// TIA Portal project "四层电梯_V17" (V17)

(* hardware
DEVICE "S7-1200 station_1"  S7-1200 Station
   slot 0: "Rack_0"  S7-1200 Rack  Rack  V1.0
   slot 1: "PLC_1"  CPU 1214C DC/DC/DC  6ES7 214-1AG40-0XB0  V4.2
DEVICE "HMI_1"  KTP700 Basic PN
   slot 0: "HMI_1"  KTP700 Basic PN  6AV2 123-2GB03-0AX0  15.0.0.0
   slot 1: "HMI_RT_1"  KTP700 Basic PN  6AV2 123-2GB03-0AX0  15.0.0.0
   slot 5: "HMI_1.IE_CP_1"  PROFINET Interface  15.0.0.0
      slot 1: "PROFINET Interface_1"  PROFINET Interface
         slot 1: "Port_1"  Port
*)

// ===== PLC "PLC_1"  CPU 1214C DC/DC/DC =====

VAR_GLOBAL   // PLC tag table "默认变量表"
   "System_Byte" AT %MB1 : Byte;
   "FirstScan" AT %M1.0 : Bool;
   "DiagStatusUpdate" AT %M1.1 : Bool;
   "AlwaysTRUE" AT %M1.2 : Bool;
   "AlwaysFALSE" AT %M1.3 : Bool;
   "Clock_Byte" AT %MB0 : Byte;
   "Clock_10Hz" AT %M0.0 : Bool;
   "Clock_5Hz" AT %M0.1 : Bool;
   "Clock_2.5Hz" AT %M0.2 : Bool;
   "Clock_2Hz" AT %M0.3 : Bool;
   "Clock_1.25Hz" AT %M0.4 : Bool;
   "Clock_1Hz" AT %M0.5 : Bool;
   "Clock_0.625Hz" AT %M0.6 : Bool;
   "Clock_0.5Hz" AT %M0.7 : Bool;
   "启动" AT %M10.0 : Bool;
   "步态0" AT %M20.0 : Bool;
   "停止" AT %M11.0 : Bool;
   "外呼四层下" AT %M100.0 : Bool;
   "电梯位置" AT %MD15 : DWord;
   "上外呼层" AT %MD20 : DWord;
   "外呼三层上" AT %M101.0 : Bool;
   "外呼二层上" AT %M102.0 : Bool;
   "外呼一层上" AT %M103.0 : Bool;
   "四层下指示灯" AT %M100.1 : Bool;
   "三层上指示灯" AT %M101.1 : Bool;
   "二层上指示灯" AT %M102.1 : Bool;
   "一层上指示灯" AT %M103.1 : Bool;
   "步态1" AT %M30.0 : Bool;
   "外呼二层下" AT %M110.0 : Bool;
   "二层下指示灯" AT %M110.1 : Bool;
   "下外呼层" AT %MD30 : DWord;
   "外呼三层下" AT %M111.0 : Bool;
   "三层下指示灯" AT %M111.1 : Bool;
   "步态2" AT %M40.0 : Bool;
   "四层内呼" AT %M120.0 : Bool;
   "四层内呼指示" AT %M120.1 : Bool;
   "内呼层" AT %MD40 : DWord;
   "三层内呼" AT %M121.0 : Bool;
   "三层内呼指示" AT %M121.1 : Bool;
   "二层内呼" AT %M122.0 : Bool;
   "二层内呼指示" AT %M122.1 : Bool;
   "一层内呼" AT %M123.0 : Bool;
   "一层内呼指示" AT %M123.1 : Bool;
   "步态3" AT %M50.0 : Bool;
   "上行" AT %M3.0 : Bool;
   "下行" AT %M3.1 : Bool;
   "开关门中" AT %M60.0 : Bool;
   "Tag_1" AT %MW10 : Word;
   "目标楼层" AT %MD50 : DWord;
   "Tag_2" AT %M112.1 : Bool;
   "Tag_3" AT %M13.1 : Bool;
   "Tag_4" AT %M45.0 : Bool;
   "Tag_5" AT %M29.0 : Bool;
   "Tag_6" AT %M19.0 : Bool;
   "Tag_7" AT %M39.0 : Bool;
   "Tag_8" AT %M2.0 : Bool;
   "Tag_9" AT %M2.1 : Bool;
   "Tag_10" AT %MD60 : UDInt;
   "实际楼层数" AT %MD70 : UDInt;
   "Tag_11" AT %M10.1 : Bool;
   "Tag_12" AT %M11.1 : Bool;
   "启动指示灯" AT %M10.2 : Bool;
   "停止指示灯" AT %M11.2 : Bool;
   "一楼开门" AT %M200.0 : Bool;
   "Tag_14" AT %M200.1 : Bool;
   "门水平移动1" AT %MD150 : DWord;
   "关门延时1" AT %M200.2 : Bool;
   "二楼开门" AT %M201.0 : Bool;
   "一楼关门" AT %M200.3 : Bool;
   "Tag_15" AT %M200.4 : Bool;
   "Tag_16" AT %M200.5 : Bool;
   "一开" AT %M200.6 : Bool;
   "三楼开门" AT %M202.0 : Bool;
   "四楼开门" AT %M203.0 : Bool;
   "Tag_13" AT %M201.1 : Bool;
   "m202.2" AT %M201.2 : Bool;
   "关门延时2" AT %M201.3 : Bool;
   "门水平移动2" AT %MD160 : DInt;
   "二关" AT %M201.4 : Bool;
   "Tag_20" AT %M201.5 : Bool;
   "Tag_21" AT %M201.6 : Bool;
   "一楼关门完成位" AT %M200.7 : Bool;
   "Tag_22" AT %M201.7 : Bool;
   "Tag_23" AT %M199.0 : Bool;
   "Tag_24" AT %M199.1 : Bool;
   "三开" AT %M202.2 : Bool;
   "门水平移动3" AT %MD170 : DInt;
   "开门延时3" AT %M202.3 : Bool;
   "Tag_18" AT %M202.5 : Bool;
   "3关" AT %M202.4 : Bool;
   "Tag_17" AT %M202.1 : Bool;
   "Tag_19" AT %M203.1 : Bool;
   "4 开" AT %M203.2 : Bool;
   "Tag_26" AT %M203.5 : Bool;
   "门水平移动4" AT %MD180 : DInt;
   "关门延时4" AT %M203.3 : Bool;
   "4关" AT %M203.4 : Bool;
   "Tag_25" AT %M202.6 : Bool;
   "Tag_27" AT %M203.6 : Bool;
END_VAR

DATA_BLOCK "开关门动画_DB_2"   // DB4
{ S7_Optimized_Access := 'TRUE' }
VERSION : 0.1
// stored: InstanceOfName 开关门动画
"开关门动画"
BEGIN
END_DATA_BLOCK

// folder: System blocks/Program resources

DATA_BLOCK "IEC_Timer_0_DB_2"   // DB1
{ S7_Optimized_Access := 'TRUE' }
AUTHOR : Simatic
FAMILY : IEC
NAME : IEC_TMR
VERSION : 1.0
// stored: InstanceOfName IEC_TIMER
"IEC_TIMER"
BEGIN
END_DATA_BLOCK

DATA_BLOCK "IEC_Timer_0_DB_1"   // DB2
{ S7_Optimized_Access := 'TRUE' }
AUTHOR : Simatic
FAMILY : IEC
NAME : IEC_TMR
VERSION : 1.0
// stored: InstanceOfName IEC_TIMER
"IEC_TIMER"
BEGIN
END_DATA_BLOCK

DATA_BLOCK "IEC_Timer_0_DB_3"   // DB3
{ S7_Optimized_Access := 'TRUE' }
AUTHOR : Simatic
FAMILY : IEC
NAME : IEC_TMR
VERSION : 1.0
// stored: InstanceOfName IEC_TIMER
"IEC_TIMER"
BEGIN
END_DATA_BLOCK

DATA_BLOCK "IEC_Timer_0_DB"   // DB5
{ S7_Optimized_Access := 'TRUE' }
AUTHOR : Simatic
FAMILY : IEC
NAME : IEC_TMR
VERSION : 1.0
// stored: InstanceOfName IEC_TIMER
"IEC_TIMER"
BEGIN
END_DATA_BLOCK

// folder: (top level)

FUNCTION_BLOCK "开关门动画"   // FB1, LAD
{ S7_Optimized_Access := 'TRUE' }
VERSION : 0.1
   VAR_TEMP   // added for the SCL form of the ladder/FBD networks
      _w1 : Bool;
      _w2 : Bool;
      _w3 : Bool;
   END_VAR
BEGIN

REGION Network 1
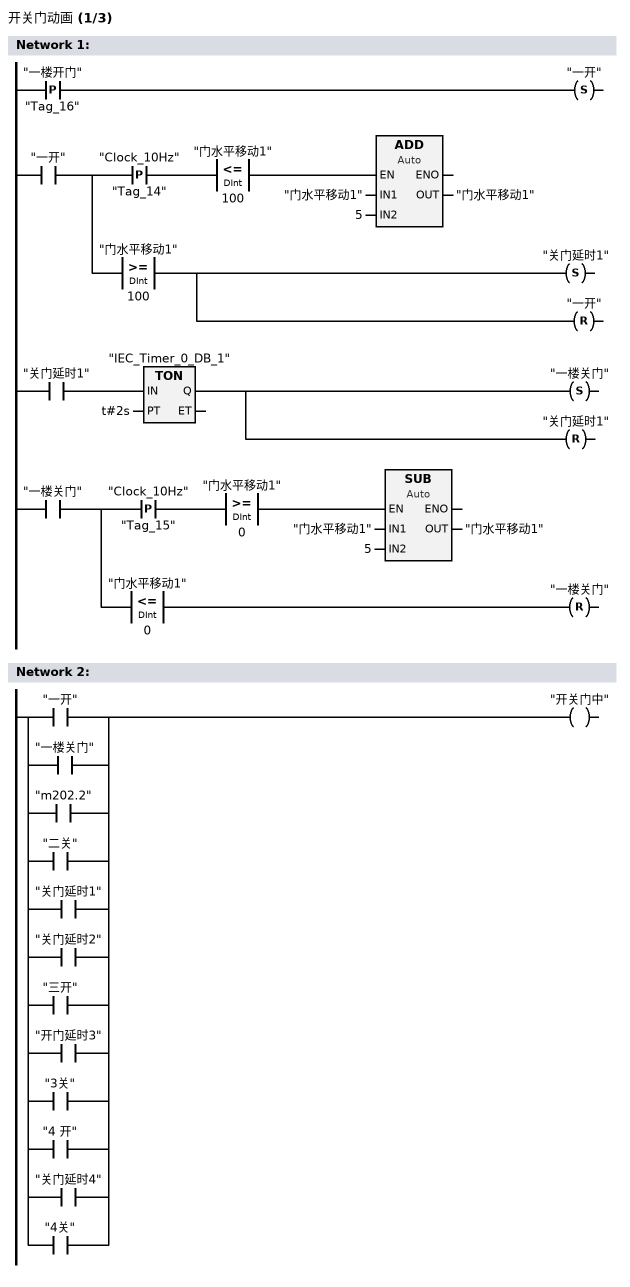
   #_w1 := "一楼开门" AND NOT "Tag_16";   // rising edge of "一楼开门"
   "Tag_16" := "一楼开门";
   IF #_w1 THEN "一开" := TRUE; END_IF;
   #_w2 := "一开" AND "Clock_10Hz" AND NOT "Tag_14";   // rising edge of "Clock_10Hz"
   "Tag_14" := "Clock_10Hz";
   IF #_w2 AND ("门水平移动1" <= 100) THEN "门水平移动1" := "门水平移动1" + 5; END_IF;
   IF "一开" AND ("门水平移动1" >= 100) THEN
       "关门延时1" := TRUE;
       "一开" := FALSE;
   END_IF;
   "IEC_Timer_0_DB_1".TON(IN := "关门延时1", PT := t#2s);
   IF "IEC_Timer_0_DB_1".Q THEN
       "一楼关门" := TRUE;
       "关门延时1" := FALSE;
   END_IF;
   #_w3 := "一楼关门" AND "Clock_10Hz" AND NOT "Tag_15";   // rising edge of "Clock_10Hz"
   "Tag_15" := "Clock_10Hz";
   IF #_w3 AND ("门水平移动1" >= 0) THEN "门水平移动1" := "门水平移动1" - 5; END_IF;
   IF "一楼关门" AND ("门水平移动1" <= 0) THEN "一楼关门" := FALSE; END_IF;
END_REGION

REGION Network 2
   RUNG wire#powerrail
      Contact( "一开" )
      wire#w1
      Coil( "开关门中" )
   END_RUNG
   RUNG wire#powerrail
      Contact( "一楼关门" )
   END_RUNG wire#w1
   RUNG wire#powerrail
      Contact( "m202.2" )
   END_RUNG wire#w1
   RUNG wire#powerrail
      Contact( "二关" )
   END_RUNG wire#w1
   RUNG wire#powerrail
      Contact( "关门延时1" )
   END_RUNG wire#w1
   RUNG wire#powerrail
      Contact( "关门延时2" )
   END_RUNG wire#w1
   RUNG wire#powerrail
      Contact( "三开" )
   END_RUNG wire#w1
   RUNG wire#powerrail
      Contact( "开门延时3" )
   END_RUNG wire#w1
   RUNG wire#powerrail
      Contact( "3关" )
   END_RUNG wire#w1
   RUNG wire#powerrail
      Contact( "4 开" )
   END_RUNG wire#w1
   RUNG wire#powerrail
      Contact( "关门延时4" )
   END_RUNG wire#w1
   RUNG wire#powerrail
      Contact( "4关" )
   END_RUNG wire#w1
   // the same network as SCL:
   "开关门中" := "一开" OR "一楼关门" OR "m202.2" OR "二关" OR "关门延时1" OR "关门延时2" OR "三开" OR "开门延时3" OR "3关" OR "4 开" OR "关门延时4" OR "4关";
END_REGION

REGION Network 3
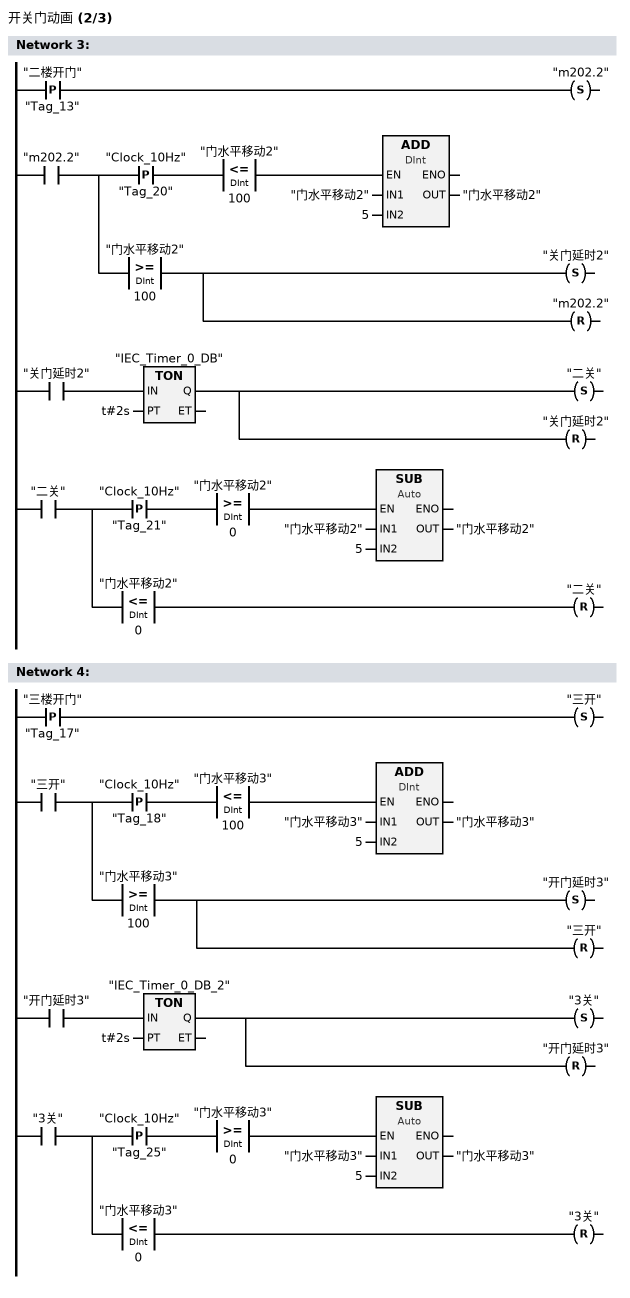
   #_w1 := "二楼开门" AND NOT "Tag_13";   // rising edge of "二楼开门"
   "Tag_13" := "二楼开门";
   IF #_w1 THEN "m202.2" := TRUE; END_IF;
   #_w2 := "m202.2" AND "Clock_10Hz" AND NOT "Tag_20";   // rising edge of "Clock_10Hz"
   "Tag_20" := "Clock_10Hz";
   IF #_w2 AND ("门水平移动2" <= 100) THEN "门水平移动2" := "门水平移动2" + 5; END_IF;
   IF "m202.2" AND ("门水平移动2" >= 100) THEN
       "关门延时2" := TRUE;
       "m202.2" := FALSE;
   END_IF;
   "IEC_Timer_0_DB".TON(IN := "关门延时2", PT := t#2s);
   IF "IEC_Timer_0_DB".Q THEN
       "二关" := TRUE;
       "关门延时2" := FALSE;
   END_IF;
   #_w3 := "二关" AND "Clock_10Hz" AND NOT "Tag_21";   // rising edge of "Clock_10Hz"
   "Tag_21" := "Clock_10Hz";
   IF #_w3 AND ("门水平移动2" >= 0) THEN "门水平移动2" := "门水平移动2" - 5; END_IF;
   IF "二关" AND ("门水平移动2" <= 0) THEN "二关" := FALSE; END_IF;
END_REGION

REGION Network 4
   #_w1 := "三楼开门" AND NOT "Tag_17";   // rising edge of "三楼开门"
   "Tag_17" := "三楼开门";
   IF #_w1 THEN "三开" := TRUE; END_IF;
   #_w2 := "三开" AND "Clock_10Hz" AND NOT "Tag_18";   // rising edge of "Clock_10Hz"
   "Tag_18" := "Clock_10Hz";
   IF #_w2 AND ("门水平移动3" <= 100) THEN "门水平移动3" := "门水平移动3" + 5; END_IF;
   IF "三开" AND ("门水平移动3" >= 100) THEN
       "开门延时3" := TRUE;
       "三开" := FALSE;
   END_IF;
   "IEC_Timer_0_DB_2".TON(IN := "开门延时3", PT := t#2s);
   IF "IEC_Timer_0_DB_2".Q THEN
       "3关" := TRUE;
       "开门延时3" := FALSE;
   END_IF;
   #_w3 := "3关" AND "Clock_10Hz" AND NOT "Tag_25";   // rising edge of "Clock_10Hz"
   "Tag_25" := "Clock_10Hz";
   IF #_w3 AND ("门水平移动3" >= 0) THEN "门水平移动3" := "门水平移动3" - 5; END_IF;
   IF "3关" AND ("门水平移动3" <= 0) THEN "3关" := FALSE; END_IF;
END_REGION

REGION Network 5
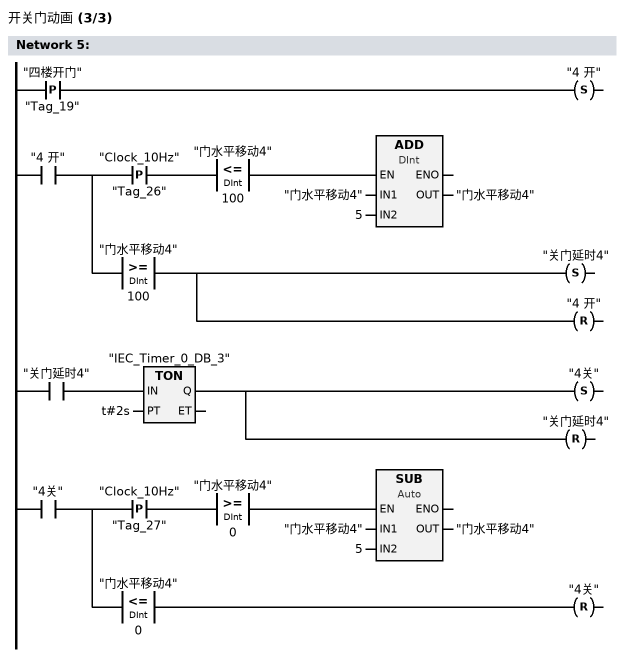
   #_w1 := "四楼开门" AND NOT "Tag_19";   // rising edge of "四楼开门"
   "Tag_19" := "四楼开门";
   IF #_w1 THEN "4 开" := TRUE; END_IF;
   #_w2 := "4 开" AND "Clock_10Hz" AND NOT "Tag_26";   // rising edge of "Clock_10Hz"
   "Tag_26" := "Clock_10Hz";
   IF #_w2 AND ("门水平移动4" <= 100) THEN "门水平移动4" := "门水平移动4" + 5; END_IF;
   IF "4 开" AND ("门水平移动4" >= 100) THEN
       "关门延时4" := TRUE;
       "4 开" := FALSE;
   END_IF;
   "IEC_Timer_0_DB_3".TON(IN := "关门延时4", PT := t#2s);
   IF "IEC_Timer_0_DB_3".Q THEN
       "4关" := TRUE;
       "关门延时4" := FALSE;
   END_IF;
   #_w3 := "4关" AND "Clock_10Hz" AND NOT "Tag_27";   // rising edge of "Clock_10Hz"
   "Tag_27" := "Clock_10Hz";
   IF #_w3 AND ("门水平移动4" >= 0) THEN "门水平移动4" := "门水平移动4" - 5; END_IF;
   IF "4关" AND ("门水平移动4" <= 0) THEN "4关" := FALSE; END_IF;
END_REGION
END_FUNCTION_BLOCK

ORGANIZATION_BLOCK "Main"   // OB1, LAD, ProgramCycle
TITLE = "Main Program Sweep (Cycle)"
{ S7_Optimized_Access := 'TRUE' }
VERSION : 0.1
   VAR_INPUT
      Initial_Call : Bool;   // Initial call of this OB
      Remanence : Bool;   // =True, if remanent data are available
   END_VAR
   VAR_TEMP   // added for the SCL form of the ladder/FBD networks
      _w1 : Bool;
      _w2 : Bool;
      _w3 : Bool;
      _w4 : Bool;
      _w5 : Bool;
   END_VAR
BEGIN

REGION Network 1
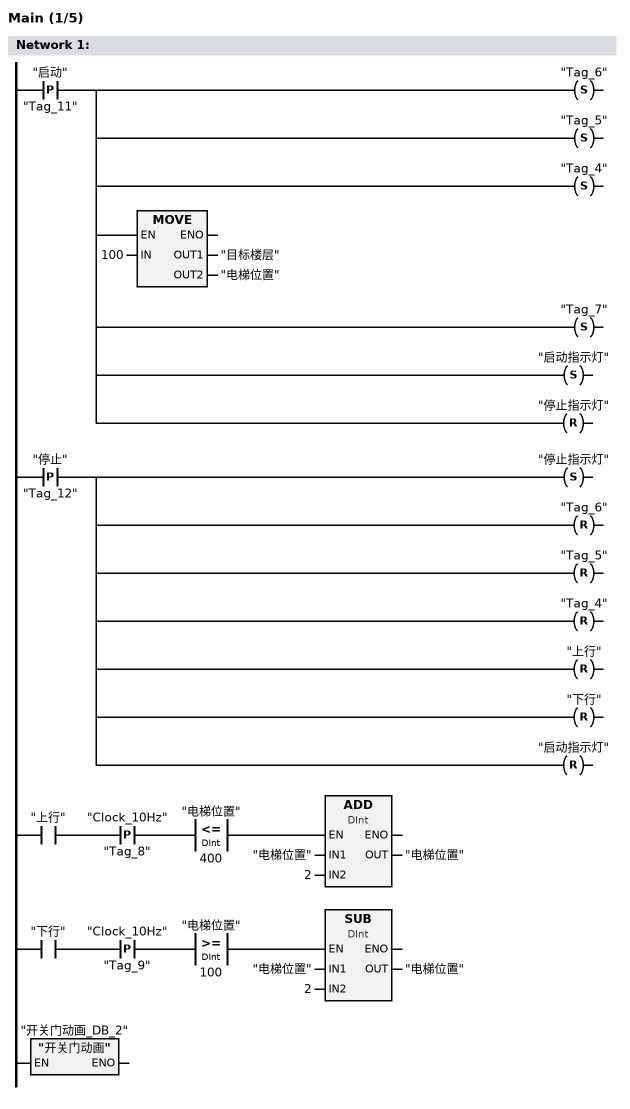
   RUNG wire#powerrail
      P_Contact(operand := "启动", bit := "Tag_11")
      wire#w1
      S_Coil( "Tag_6" )
   END_RUNG
   RUNG wire#w1
      S_Coil( "Tag_5" )
   END_RUNG
   RUNG wire#w1
      S_Coil( "Tag_4" )
   END_RUNG
   RUNG wire#w1
      Move(in := 100, out1 => "目标楼层", out2 => "电梯位置")
   END_RUNG
   RUNG wire#w1
      S_Coil( "Tag_7" )
   END_RUNG
   RUNG wire#w1
      S_Coil( "启动指示灯" )
   END_RUNG
   RUNG wire#w1
      R_Coil( "停止指示灯" )
   END_RUNG
   RUNG wire#powerrail
      P_Contact(operand := "停止", bit := "Tag_12")
      wire#w2
      S_Coil( "停止指示灯" )
   END_RUNG
   RUNG wire#w2
      R_Coil( "Tag_6" )
   END_RUNG
   RUNG wire#w2
      R_Coil( "Tag_5" )
   END_RUNG
   RUNG wire#w2
      R_Coil( "Tag_4" )
   END_RUNG
   RUNG wire#w2
      R_Coil( "上行" )
   END_RUNG
   RUNG wire#w2
      R_Coil( "下行" )
   END_RUNG
   RUNG wire#w2
      R_Coil( "启动指示灯" )
   END_RUNG
   RUNG wire#powerrail
      Contact( "上行" )
      P_Contact(operand := "Clock_10Hz", bit := "Tag_8")
      { S7_Templates := "SrcType := DInt" } LE_Contact(in1 := "电梯位置", in2 := 400)
      { S7_Templates := "SrcType := DInt" } Add(in1 := "电梯位置", in2 := 2, out => "电梯位置")
   END_RUNG
   RUNG wire#powerrail
      Contact( "下行" )
      P_Contact(operand := "Clock_10Hz", bit := "Tag_9")
      { S7_Templates := "SrcType := DInt" } GE_Contact(in1 := "电梯位置", in2 := 100)
      { S7_Templates := "SrcType := DInt" } Sub(in1 := "电梯位置", in2 := 2, out => "电梯位置")
   END_RUNG
   RUNG wire#powerrail
      "开关门动画_DB_2"()
   END_RUNG
   // the same network as SCL:
   #_w1 := "启动" AND NOT "Tag_11";   // rising edge of "启动"
   "Tag_11" := "启动";
   IF #_w1 THEN
       "Tag_6" := TRUE;
       "Tag_5" := TRUE;
       "Tag_4" := TRUE;
       "目标楼层" := 100;
       "电梯位置" := 100;
       "Tag_7" := TRUE;
       "启动指示灯" := TRUE;
       "停止指示灯" := FALSE;
   END_IF;
   #_w2 := "停止" AND NOT "Tag_12";   // rising edge of "停止"
   "Tag_12" := "停止";
   IF #_w2 THEN
       "停止指示灯" := TRUE;
       "Tag_6" := FALSE;
       "Tag_5" := FALSE;
       "Tag_4" := FALSE;
       "上行" := FALSE;
       "下行" := FALSE;
       "启动指示灯" := FALSE;
   END_IF;
   #_w3 := "上行" AND "Clock_10Hz" AND NOT "Tag_8";   // rising edge of "Clock_10Hz"
   "Tag_8" := "Clock_10Hz";
   IF #_w3 AND ("电梯位置" <= 400) THEN "电梯位置" := "电梯位置" + 2; END_IF;
   #_w4 := "下行" AND "Clock_10Hz" AND NOT "Tag_9";   // rising edge of "Clock_10Hz"
   "Tag_9" := "Clock_10Hz";
   IF #_w4 AND ("电梯位置" >= 100) THEN "电梯位置" := "电梯位置" - 2; END_IF;
   "开关门动画_DB_2"();   // "开关门动画"
END_REGION

REGION Network 2: 外呼上采集
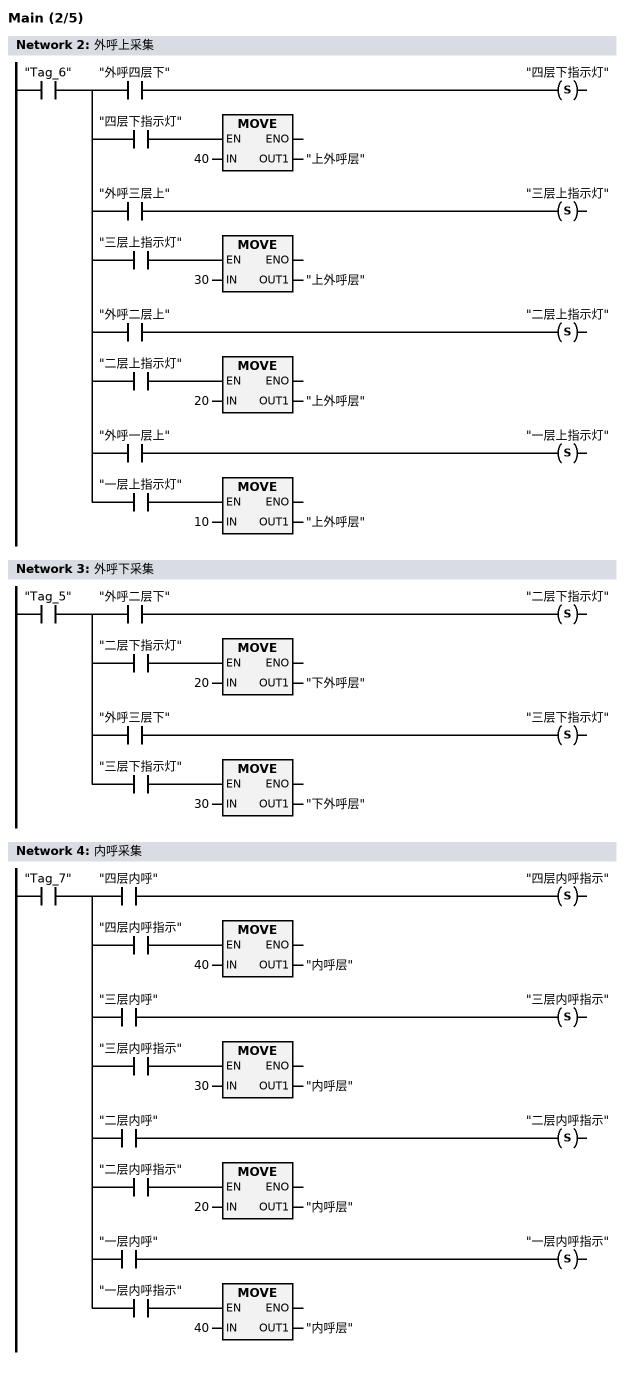
   RUNG wire#powerrail
      Contact( "Tag_6" )
      wire#w1
      Contact( "外呼四层下" )
      S_Coil( "四层下指示灯" )
   END_RUNG
   RUNG wire#w1
      Contact( "四层下指示灯" )
      Move(in := 40, out1 => "上外呼层")
   END_RUNG
   RUNG wire#w1
      Contact( "外呼三层上" )
      S_Coil( "三层上指示灯" )
   END_RUNG
   RUNG wire#w1
      Contact( "三层上指示灯" )
      Move(in := 30, out1 => "上外呼层")
   END_RUNG
   RUNG wire#w1
      Contact( "外呼二层上" )
      S_Coil( "二层上指示灯" )
   END_RUNG
   RUNG wire#w1
      Contact( "二层上指示灯" )
      Move(in := 20, out1 => "上外呼层")
   END_RUNG
   RUNG wire#w1
      Contact( "外呼一层上" )
      S_Coil( "一层上指示灯" )
   END_RUNG
   RUNG wire#w1
      Contact( "一层上指示灯" )
      Move(in := 10, out1 => "上外呼层")
   END_RUNG
   // the same network as SCL:
   IF "Tag_6" AND "外呼四层下" THEN "四层下指示灯" := TRUE; END_IF;
   IF "Tag_6" AND "四层下指示灯" THEN "上外呼层" := 40; END_IF;
   IF "Tag_6" AND "外呼三层上" THEN "三层上指示灯" := TRUE; END_IF;
   IF "Tag_6" AND "三层上指示灯" THEN "上外呼层" := 30; END_IF;
   IF "Tag_6" AND "外呼二层上" THEN "二层上指示灯" := TRUE; END_IF;
   IF "Tag_6" AND "二层上指示灯" THEN "上外呼层" := 20; END_IF;
   IF "Tag_6" AND "外呼一层上" THEN "一层上指示灯" := TRUE; END_IF;
   IF "Tag_6" AND "一层上指示灯" THEN "上外呼层" := 10; END_IF;
END_REGION

REGION Network 3: 外呼下采集
   RUNG wire#powerrail
      Contact( "Tag_5" )
      wire#w1
      Contact( "外呼二层下" )
      S_Coil( "二层下指示灯" )
   END_RUNG
   RUNG wire#w1
      Contact( "二层下指示灯" )
      Move(in := 20, out1 => "下外呼层")
   END_RUNG
   RUNG wire#w1
      Contact( "外呼三层下" )
      S_Coil( "三层下指示灯" )
   END_RUNG
   RUNG wire#w1
      Contact( "三层下指示灯" )
      Move(in := 30, out1 => "下外呼层")
   END_RUNG
   // the same network as SCL:
   IF "Tag_5" AND "外呼二层下" THEN "二层下指示灯" := TRUE; END_IF;
   IF "Tag_5" AND "二层下指示灯" THEN "下外呼层" := 20; END_IF;
   IF "Tag_5" AND "外呼三层下" THEN "三层下指示灯" := TRUE; END_IF;
   IF "Tag_5" AND "三层下指示灯" THEN "下外呼层" := 30; END_IF;
END_REGION

REGION Network 4: 内呼采集
   RUNG wire#powerrail
      Contact( "Tag_7" )
      wire#w1
      Contact( "四层内呼" )
      S_Coil( "四层内呼指示" )
   END_RUNG
   RUNG wire#w1
      Contact( "四层内呼指示" )
      Move(in := 40, out1 => "内呼层")
   END_RUNG
   RUNG wire#w1
      Contact( "三层内呼" )
      S_Coil( "三层内呼指示" )
   END_RUNG
   RUNG wire#w1
      Contact( "三层内呼指示" )
      Move(in := 30, out1 => "内呼层")
   END_RUNG
   RUNG wire#w1
      Contact( "二层内呼" )
      S_Coil( "二层内呼指示" )
   END_RUNG
   RUNG wire#w1
      Contact( "二层内呼指示" )
      Move(in := 20, out1 => "内呼层")
   END_RUNG
   RUNG wire#w1
      Contact( "一层内呼" )
      S_Coil( "一层内呼指示" )
   END_RUNG
   RUNG wire#w1
      Contact( "一层内呼指示" )
      Move(in := 40, out1 => "内呼层")
   END_RUNG
   // the same network as SCL:
   IF "Tag_7" AND "四层内呼" THEN "四层内呼指示" := TRUE; END_IF;
   IF "Tag_7" AND "四层内呼指示" THEN "内呼层" := 40; END_IF;
   IF "Tag_7" AND "三层内呼" THEN "三层内呼指示" := TRUE; END_IF;
   IF "Tag_7" AND "三层内呼指示" THEN "内呼层" := 30; END_IF;
   IF "Tag_7" AND "二层内呼" THEN "二层内呼指示" := TRUE; END_IF;
   IF "Tag_7" AND "二层内呼指示" THEN "内呼层" := 20; END_IF;
   IF "Tag_7" AND "一层内呼" THEN "一层内呼指示" := TRUE; END_IF;
   IF "Tag_7" AND "一层内呼指示" THEN "内呼层" := 40; END_IF;
END_REGION

REGION Network 5: 上行需求响应
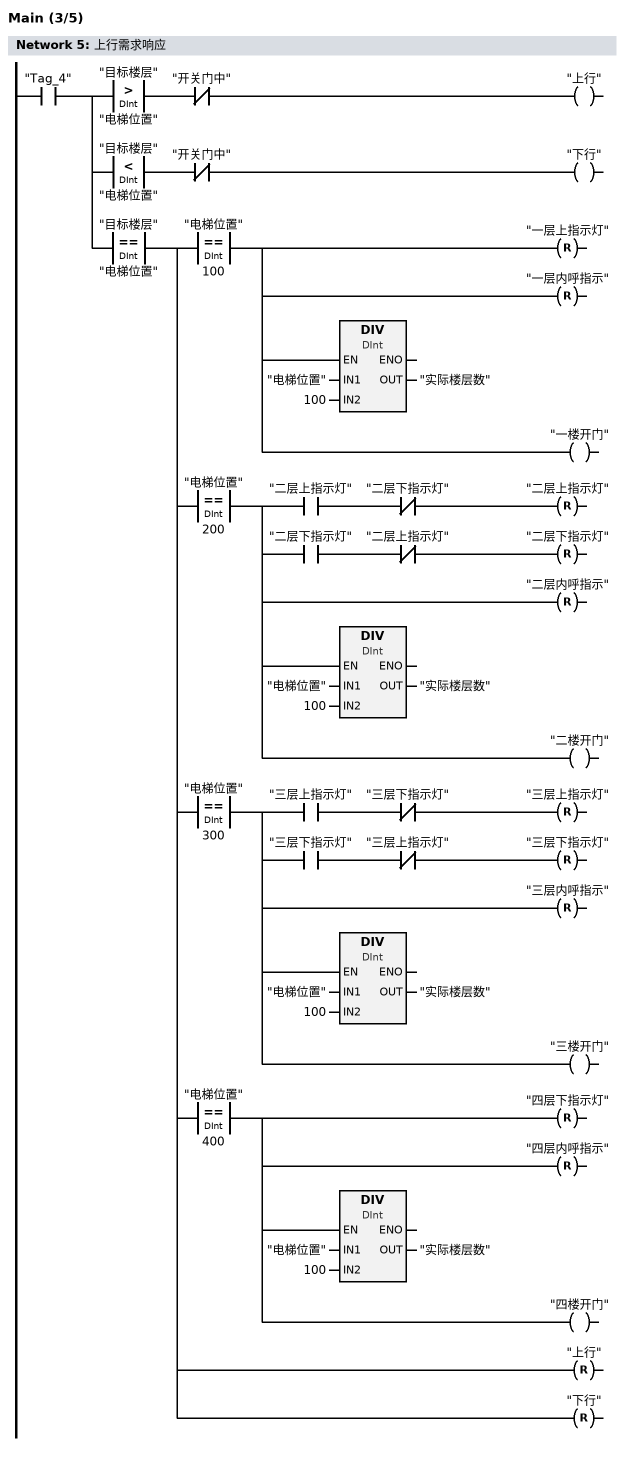
   RUNG wire#powerrail
      Contact( "Tag_4" )
      wire#w1
      { S7_Templates := "SrcType := DInt" } GT_Contact(in1 := "目标楼层", in2 := "电梯位置")
      I_Contact( "开关门中" )
      Coil( "上行" )
   END_RUNG
   RUNG wire#w1
      { S7_Templates := "SrcType := DInt" } LT_Contact(in1 := "目标楼层", in2 := "电梯位置")
      I_Contact( "开关门中" )
      Coil( "下行" )
   END_RUNG
   RUNG wire#w1
      { S7_Templates := "SrcType := DInt" } EQ_Contact(in1 := "目标楼层", in2 := "电梯位置")
      wire#w2
      { S7_Templates := "SrcType := DInt" } EQ_Contact(in1 := "电梯位置", in2 := 100)
      wire#w3
      R_Coil( "一层上指示灯" )
   END_RUNG
   RUNG wire#w3
      R_Coil( "一层内呼指示" )
   END_RUNG
   RUNG wire#w3
      { S7_Templates := "SrcType := DInt" } Div(in1 := "电梯位置", in2 := 100, out => "实际楼层数")
   END_RUNG
   RUNG wire#w3
      Coil( "一楼开门" )
   END_RUNG
   RUNG wire#w2
      { S7_Templates := "SrcType := DInt" } EQ_Contact(in1 := "电梯位置", in2 := 200)
      wire#w4
      Contact( "二层上指示灯" )
      I_Contact( "二层下指示灯" )
      R_Coil( "二层上指示灯" )
   END_RUNG
   RUNG wire#w4
      Contact( "二层下指示灯" )
      I_Contact( "二层上指示灯" )
      R_Coil( "二层下指示灯" )
   END_RUNG
   RUNG wire#w4
      R_Coil( "二层内呼指示" )
   END_RUNG
   RUNG wire#w4
      { S7_Templates := "SrcType := DInt" } Div(in1 := "电梯位置", in2 := 100, out => "实际楼层数")
   END_RUNG
   RUNG wire#w4
      Coil( "二楼开门" )
   END_RUNG
   RUNG wire#w2
      { S7_Templates := "SrcType := DInt" } EQ_Contact(in1 := "电梯位置", in2 := 300)
      wire#w5
      Contact( "三层上指示灯" )
      I_Contact( "三层下指示灯" )
      R_Coil( "三层上指示灯" )
   END_RUNG
   RUNG wire#w5
      Contact( "三层下指示灯" )
      I_Contact( "三层上指示灯" )
      R_Coil( "三层下指示灯" )
   END_RUNG
   RUNG wire#w5
      R_Coil( "三层内呼指示" )
   END_RUNG
   RUNG wire#w5
      { S7_Templates := "SrcType := DInt" } Div(in1 := "电梯位置", in2 := 100, out => "实际楼层数")
   END_RUNG
   RUNG wire#w5
      Coil( "三楼开门" )
   END_RUNG
   RUNG wire#w2
      { S7_Templates := "SrcType := DInt" } EQ_Contact(in1 := "电梯位置", in2 := 400)
      wire#w6
      R_Coil( "四层下指示灯" )
   END_RUNG
   RUNG wire#w6
      R_Coil( "四层内呼指示" )
   END_RUNG
   RUNG wire#w6
      { S7_Templates := "SrcType := DInt" } Div(in1 := "电梯位置", in2 := 100, out => "实际楼层数")
   END_RUNG
   RUNG wire#w6
      Coil( "四楼开门" )
   END_RUNG
   RUNG wire#w2
      R_Coil( "上行" )
   END_RUNG
   RUNG wire#w2
      R_Coil( "下行" )
   END_RUNG
   // the same network as SCL:
   "上行" := "Tag_4" AND ("目标楼层" > "电梯位置") AND NOT "开关门中";
   "下行" := "Tag_4" AND ("目标楼层" < "电梯位置") AND NOT "开关门中";
   #_w1 := "Tag_4" AND ("目标楼层" = "电梯位置");
   #_w2 := #_w1 AND ("电梯位置" = 100);
   IF #_w2 THEN
       "一层上指示灯" := FALSE;
       "一层内呼指示" := FALSE;
       "实际楼层数" := "电梯位置" / 100;
   END_IF;
   "一楼开门" := #_w2;
   #_w3 := #_w1 AND ("电梯位置" = 200);
   IF #_w3 AND "二层上指示灯" AND NOT "二层下指示灯" THEN "二层上指示灯" := FALSE; END_IF;
   IF #_w3 AND "二层下指示灯" AND NOT "二层上指示灯" THEN "二层下指示灯" := FALSE; END_IF;
   IF #_w3 THEN
       "二层内呼指示" := FALSE;
       "实际楼层数" := "电梯位置" / 100;
   END_IF;
   "二楼开门" := #_w3;
   #_w4 := #_w1 AND ("电梯位置" = 300);
   IF #_w4 AND "三层上指示灯" AND NOT "三层下指示灯" THEN "三层上指示灯" := FALSE; END_IF;
   IF #_w4 AND "三层下指示灯" AND NOT "三层上指示灯" THEN "三层下指示灯" := FALSE; END_IF;
   IF #_w4 THEN
       "三层内呼指示" := FALSE;
       "实际楼层数" := "电梯位置" / 100;
   END_IF;
   "三楼开门" := #_w4;
   #_w5 := #_w1 AND ("电梯位置" = 400);
   IF #_w5 THEN
       "四层下指示灯" := FALSE;
       "四层内呼指示" := FALSE;
       "实际楼层数" := "电梯位置" / 100;
   END_IF;
   "四楼开门" := #_w5;
   IF #_w1 THEN
       "上行" := FALSE;
       "下行" := FALSE;
   END_IF;
END_REGION

REGION Network 6: 开门延时
END_REGION

REGION Network 7: 在一楼判断目标楼层
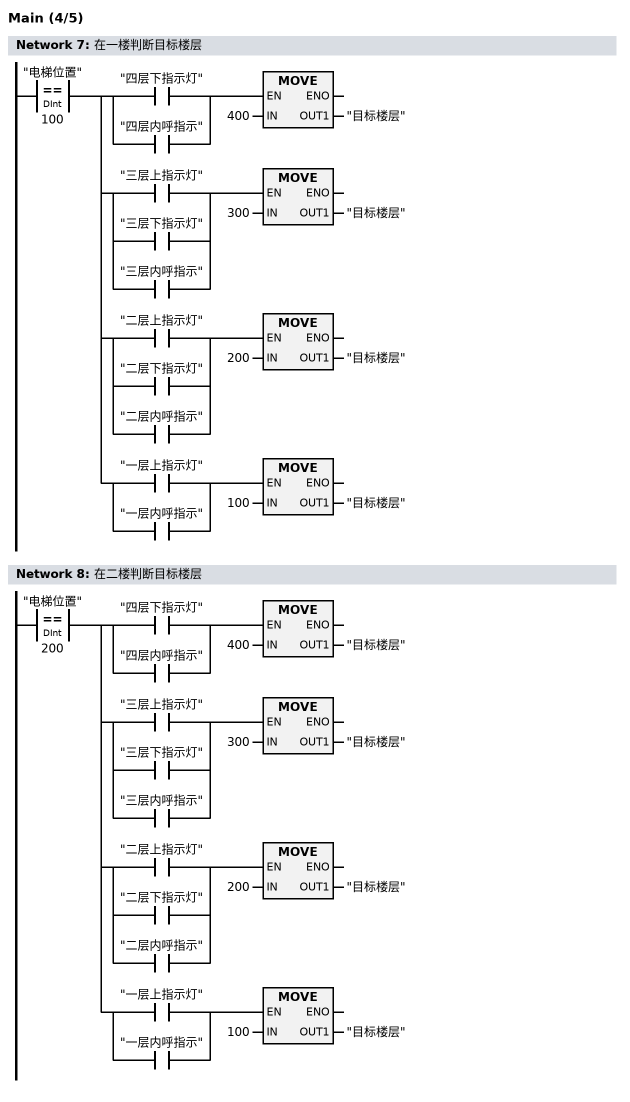
   RUNG wire#powerrail
      { S7_Templates := "SrcType := DInt" } EQ_Contact(in1 := "电梯位置", in2 := 100)
      wire#w1
      Contact( "四层下指示灯" )
      wire#w2
      Move(in := 400, out1 => "目标楼层")
   END_RUNG
   RUNG wire#w1
      Contact( "四层内呼指示" )
   END_RUNG wire#w2
   RUNG wire#w1
      Contact( "三层上指示灯" )
      wire#w3
      Move(in := 300, out1 => "目标楼层")
   END_RUNG
   RUNG wire#w1
      Contact( "三层下指示灯" )
   END_RUNG wire#w3
   RUNG wire#w1
      Contact( "三层内呼指示" )
   END_RUNG wire#w3
   RUNG wire#w1
      Contact( "二层上指示灯" )
      wire#w4
      Move(in := 200, out1 => "目标楼层")
   END_RUNG
   RUNG wire#w1
      Contact( "二层下指示灯" )
   END_RUNG wire#w4
   RUNG wire#w1
      Contact( "二层内呼指示" )
   END_RUNG wire#w4
   RUNG wire#w1
      Contact( "一层上指示灯" )
      wire#w5
      Move(in := 100, out1 => "目标楼层")
   END_RUNG
   RUNG wire#w1
      Contact( "一层内呼指示" )
   END_RUNG wire#w5
   // the same network as SCL:
   #_w1 := "电梯位置" = 100;
   IF #_w1 AND ("四层下指示灯" OR "四层内呼指示") THEN "目标楼层" := 400; END_IF;
   IF #_w1 AND ("三层上指示灯" OR "三层下指示灯" OR "三层内呼指示") THEN "目标楼层" := 300; END_IF;
   IF #_w1 AND ("二层上指示灯" OR "二层下指示灯" OR "二层内呼指示") THEN "目标楼层" := 200; END_IF;
   IF #_w1 AND ("一层上指示灯" OR "一层内呼指示") THEN "目标楼层" := 100; END_IF;
END_REGION

REGION Network 8: 在二楼判断目标楼层
   RUNG wire#powerrail
      { S7_Templates := "SrcType := DInt" } EQ_Contact(in1 := "电梯位置", in2 := 200)
      wire#w1
      Contact( "四层下指示灯" )
      wire#w2
      Move(in := 400, out1 => "目标楼层")
   END_RUNG
   RUNG wire#w1
      Contact( "四层内呼指示" )
   END_RUNG wire#w2
   RUNG wire#w1
      Contact( "三层上指示灯" )
      wire#w3
      Move(in := 300, out1 => "目标楼层")
   END_RUNG
   RUNG wire#w1
      Contact( "三层下指示灯" )
   END_RUNG wire#w3
   RUNG wire#w1
      Contact( "三层内呼指示" )
   END_RUNG wire#w3
   RUNG wire#w1
      Contact( "二层上指示灯" )
      wire#w4
      Move(in := 200, out1 => "目标楼层")
   END_RUNG
   RUNG wire#w1
      Contact( "二层下指示灯" )
   END_RUNG wire#w4
   RUNG wire#w1
      Contact( "二层内呼指示" )
   END_RUNG wire#w4
   RUNG wire#w1
      Contact( "一层上指示灯" )
      wire#w5
      Move(in := 100, out1 => "目标楼层")
   END_RUNG
   RUNG wire#w1
      Contact( "一层内呼指示" )
   END_RUNG wire#w5
   // the same network as SCL:
   #_w1 := "电梯位置" = 200;
   IF #_w1 AND ("四层下指示灯" OR "四层内呼指示") THEN "目标楼层" := 400; END_IF;
   IF #_w1 AND ("三层上指示灯" OR "三层下指示灯" OR "三层内呼指示") THEN "目标楼层" := 300; END_IF;
   IF #_w1 AND ("二层上指示灯" OR "二层下指示灯" OR "二层内呼指示") THEN "目标楼层" := 200; END_IF;
   IF #_w1 AND ("一层上指示灯" OR "一层内呼指示") THEN "目标楼层" := 100; END_IF;
END_REGION

REGION Network 9: 在三楼判断目标楼层
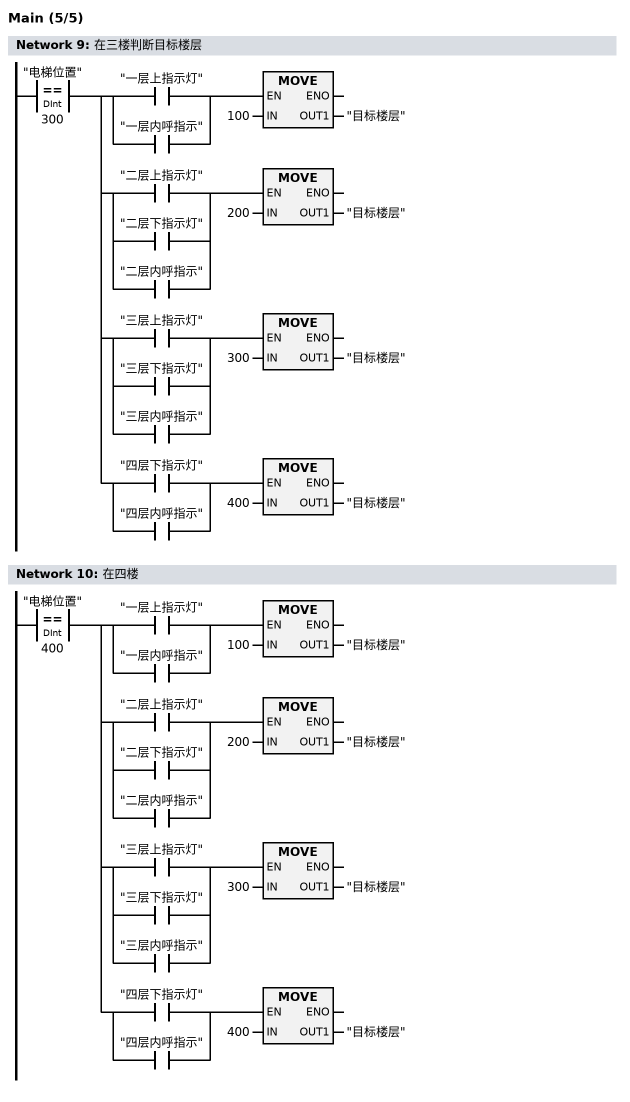
   RUNG wire#powerrail
      { S7_Templates := "SrcType := DInt" } EQ_Contact(in1 := "电梯位置", in2 := 300)
      wire#w1
      Contact( "一层上指示灯" )
      wire#w2
      Move(in := 100, out1 => "目标楼层")
   END_RUNG
   RUNG wire#w1
      Contact( "一层内呼指示" )
   END_RUNG wire#w2
   RUNG wire#w1
      Contact( "二层上指示灯" )
      wire#w3
      Move(in := 200, out1 => "目标楼层")
   END_RUNG
   RUNG wire#w1
      Contact( "二层下指示灯" )
   END_RUNG wire#w3
   RUNG wire#w1
      Contact( "二层内呼指示" )
   END_RUNG wire#w3
   RUNG wire#w1
      Contact( "三层上指示灯" )
      wire#w4
      Move(in := 300, out1 => "目标楼层")
   END_RUNG
   RUNG wire#w1
      Contact( "三层下指示灯" )
   END_RUNG wire#w4
   RUNG wire#w1
      Contact( "三层内呼指示" )
   END_RUNG wire#w4
   RUNG wire#w1
      Contact( "四层下指示灯" )
      wire#w5
      Move(in := 400, out1 => "目标楼层")
   END_RUNG
   RUNG wire#w1
      Contact( "四层内呼指示" )
   END_RUNG wire#w5
   // the same network as SCL:
   #_w1 := "电梯位置" = 300;
   IF #_w1 AND ("一层上指示灯" OR "一层内呼指示") THEN "目标楼层" := 100; END_IF;
   IF #_w1 AND ("二层上指示灯" OR "二层下指示灯" OR "二层内呼指示") THEN "目标楼层" := 200; END_IF;
   IF #_w1 AND ("三层上指示灯" OR "三层下指示灯" OR "三层内呼指示") THEN "目标楼层" := 300; END_IF;
   IF #_w1 AND ("四层下指示灯" OR "四层内呼指示") THEN "目标楼层" := 400; END_IF;
END_REGION

REGION Network 10: 在四楼
   RUNG wire#powerrail
      { S7_Templates := "SrcType := DInt" } EQ_Contact(in1 := "电梯位置", in2 := 400)
      wire#w1
      Contact( "一层上指示灯" )
      wire#w2
      Move(in := 100, out1 => "目标楼层")
   END_RUNG
   RUNG wire#w1
      Contact( "一层内呼指示" )
   END_RUNG wire#w2
   RUNG wire#w1
      Contact( "二层上指示灯" )
      wire#w3
      Move(in := 200, out1 => "目标楼层")
   END_RUNG
   RUNG wire#w1
      Contact( "二层下指示灯" )
   END_RUNG wire#w3
   RUNG wire#w1
      Contact( "二层内呼指示" )
   END_RUNG wire#w3
   RUNG wire#w1
      Contact( "三层上指示灯" )
      wire#w4
      Move(in := 300, out1 => "目标楼层")
   END_RUNG
   RUNG wire#w1
      Contact( "三层下指示灯" )
   END_RUNG wire#w4
   RUNG wire#w1
      Contact( "三层内呼指示" )
   END_RUNG wire#w4
   RUNG wire#w1
      Contact( "四层下指示灯" )
      wire#w5
      Move(in := 400, out1 => "目标楼层")
   END_RUNG
   RUNG wire#w1
      Contact( "四层内呼指示" )
   END_RUNG wire#w5
   // the same network as SCL:
   #_w1 := "电梯位置" = 400;
   IF #_w1 AND ("一层上指示灯" OR "一层内呼指示") THEN "目标楼层" := 100; END_IF;
   IF #_w1 AND ("二层上指示灯" OR "二层下指示灯" OR "二层内呼指示") THEN "目标楼层" := 200; END_IF;
   IF #_w1 AND ("三层上指示灯" OR "三层下指示灯" OR "三层内呼指示") THEN "目标楼层" := 300; END_IF;
   IF #_w1 AND ("四层下指示灯" OR "四层内呼指示") THEN "目标楼层" := 400; END_IF;
END_REGION
END_ORGANIZATION_BLOCK

(* ===== HMI "HMI_RT_1" =====
system functions are stored by id; their names below are inferred from use
connection "HMI_连接_1": ETHERNET, SMART_S7_1200_OMS

HMI tags "默认变量表"
   "Tag_ScreenNumber" : UInt, internal
   "电梯位置" : DWord = PLC 电梯位置 AT %MD15, 100 ms
   "上行" : Bool = PLC 上行 AT %M3.0, 100 ms
   "下行" : Bool = PLC 下行 AT %M3.1, 100 ms
   "外呼一层上" : Bool = PLC 外呼一层上 AT %M103.0, 100 ms
   "外呼二层上" : Bool = PLC 外呼二层上 AT %M102.0, 100 ms
   "外呼二层下" : Bool = PLC 外呼二层下 AT %M110.0, 100 ms
   "外呼三层上" : Bool = PLC 外呼三层上 AT %M101.0, 100 ms
   "外呼三层下" : Bool = PLC 外呼三层下 AT %M111.0, 100 ms
   "外呼四层下" : Bool = PLC 外呼四层下 AT %M100.0, 100 ms
   "四层下指示灯" : Bool = PLC 四层下指示灯 AT %M100.1, 100 ms
   "三层上指示灯" : Bool = PLC 三层上指示灯 AT %M101.1, 100 ms
   "三层下指示灯" : Bool = PLC 三层下指示灯 AT %M111.1, 100 ms
   "二层上指示灯" : Bool = PLC 二层上指示灯 AT %M102.1, 100 ms
   "二层下指示灯" : Bool = PLC 二层下指示灯 AT %M110.1, 100 ms
   "一层上指示灯" : Bool = PLC 一层上指示灯 AT %M103.1, 100 ms
   "四层内呼指示" : Bool = PLC 四层内呼指示 AT %M120.1, 100 ms
   "三层内呼指示" : Bool = PLC 三层内呼指示 AT %M121.1, 100 ms
   "四层内呼" : Bool = PLC 四层内呼 AT %M120.0, 100 ms
   "二层内呼指示" : Bool = PLC 二层内呼指示 AT %M122.1, 100 ms
   "一层内呼指示" : Bool = PLC 一层内呼指示 AT %M123.1, 100 ms
   "三层内呼" : Bool = PLC 三层内呼 AT %M121.0, 100 ms
   "二层内呼" : Bool = PLC 二层内呼 AT %M122.0, 100 ms
   "一层内呼" : Bool = PLC 一层内呼 AT %M123.0, 100 ms
   "实际楼层数" : UDInt = PLC 实际楼层数 AT %MD70, 100 ms
   "开门步" : Bool = PLC 开关门中 AT %M60.0, 100 ms
   "启动指示灯" : Bool = PLC 启动指示灯 AT %M10.2, 100 ms
   "停止指示灯" : Bool = PLC 停止指示灯 AT %M11.2, 100 ms
   "启动" : Bool = PLC 启动 AT %M10.0, 100 ms
   "停止" : Bool = PLC 停止 AT %M11.0, 100 ms
   "门水平移动1" : DWord = PLC 门水平移动1 AT %MD150, 100 ms
   "门水平移动2" : DInt = PLC 门水平移动2 AT %MD160, 100 ms
   "门水平移动3" : DInt = PLC 门水平移动3 AT %MD170, 100 ms
   "门水平移动4" : DInt = PLC 门水平移动4 AT %MD180, 100 ms

Template "Template_1" 800x480
   Button "Template_Button" at 714,429 size 71x50; TextOff 'Text'
   Button "Template_Button_1" at 614,429 size 71x50; TextOff 'Text'
   Button "Template_Button_2" at 514,429 size 71x50; TextOff 'Text'
   Button "Template_Button_3" at 414,429 size 71x50; TextOff 'Text'
   Button "Template_Button_4" at 314,429 size 71x50; TextOff 'Text'
   Button "Template_Button_5" at 214,429 size 71x50; TextOff 'Text'
   Button "报警" at 114,429 size 71x50; TextOff '报警'; PictureOff "AlarmDisplay_KTP700_Basic_PN_TR"; PictureOn "AlarmDisplay_KTP700_Basic_PN_TR"
      on Release: function_ef3f5d25("报警窗口_Unacknowledged", -1)
   Button "Template_Button_6" at 14,429 size 71x50; TextOff 'Text'
   SymbolicIOField "Symbolic_IO_Field_Screen" at 93,9 size 600x33; TextOff '0'; TextOn '1'; TextList "TextList_ScreenNames"
      ProcessValue <- "Tag_ScreenNumber"
      on Change: ActivateScreenByNumber("Tag_ScreenNumber", 0)
   DateTimeField "HmiScreenItemData" at 695,25 size 105x25
   DateTimeField "HmiScreenItemData_1" at 695,0 size 105x25
   GraphicView "Logo" at 0,0 size 91x51; Picture "HMI_1 的 Logo"

screen "画面_1" 800x480
   Button "按钮_1" at 722,364 size 64x44; TextOff '手动上行'
      on Press: SetBit("上行")
      on Release: ResetBit("上行")
   Button "按钮_2" at 721,419 size 68x46; TextOff '手动下行'
      on Release: ResetBit("下行")
      on Press: SetBit("下行")
   TextField "文本域_1" at 10,412 size 71x37; Text '一楼'
   TextField "文本域_2" at 10,288 size 71x37; Text '二楼'
   TextField "文本域_3" at 10,159 size 71x37; Text '三楼'
   TextField "文本域_4" at 10,31 size 71x37; Text '四楼'
   Button "按钮_3" at 262,415 size 66x34; TextOff '一楼上'
      on Press: SetBit("外呼一层上")
      on Release: ResetBit("外呼一层上")
   Button "按钮_4" at 251,283 size 66x34; TextOff '二楼上'
      on Release: ResetBit("外呼二层上")
      on Press: SetBit("外呼二层上")
   Button "按钮_5" at 339,283 size 66x34; TextOff '二楼下'
      on Release: ResetBit("外呼二层下")
      on Press: SetBit("外呼二层下")
   Button "按钮_6" at 251,156 size 66x34; TextOff '三楼上'
      on Release: ResetBit("外呼三层上")
      on Press: SetBit("外呼三层上")
   Button "按钮_7" at 340,156 size 66x34; TextOff '三楼下'
      on Release: ResetBit("外呼三层下")
      on Press: SetBit("外呼三层下")
   Button "按钮_8" at 253,26 size 66x34; TextOff '四楼下'
      on Release: ResetBit("外呼四层下")
      on Press: SetBit("外呼四层下")
   TextField "文本域_5" at 531,60 size 153x40; Text '内选按钮'
   Button "按钮_9" at 543,113 size 67x41; TextOff '4'
      on Press: SetBit("四层内呼")
      on Release: ResetBit("四层内呼")
   Circle "圆_1" at 332,26 size 33x33
      Appearance <- "四层下指示灯"
   Circle "圆_2" at 265,189 size 33x33
      Appearance <- "三层上指示灯"
   Circle "圆_3" at 355,187 size 33x33
      Appearance <- "三层下指示灯"
   Circle "圆_4" at 626,113 size 33x33
      Appearance <- "四层内呼指示"
   Circle "圆_5" at 626,170 size 33x33
      Appearance <- "三层内呼指示"
   Circle "圆_6" at 626,226 size 33x33
      Appearance <- "二层内呼指示"
   Circle "圆_7" at 626,278 size 33x33
      Appearance <- "一层内呼指示"
   Circle "圆_8" at 269,317 size 33x33
      Appearance <- "二层上指示灯"
   Circle "圆_9" at 356,317 size 33x33
      Appearance <- "二层下指示灯"
   Circle "圆_10" at 340,415 size 33x33
      Appearance <- "一层上指示灯"
   Button "按钮_10" at 543,167 size 67x41; TextOff '3'
      on Release: ResetBit("三层内呼")
      on Press: SetBit("三层内呼")
   Button "按钮_11" at 542,224 size 67x41; TextOff '2'
      on Release: ResetBit("二层内呼")
      on Press: SetBit("二层内呼")
   Button "按钮_12" at 543,275 size 67x41; TextOff '1'
      on Release: ResetBit("一层内呼")
      on Press: SetBit("一层内呼")
   TextField "文本域_6" at 495,6 size 153x40; Text '开关门中'
   IOField "I/O 域_1" at 538,324 size 63x84; FormatPattern 9
      ProcessValue <- "实际楼层数"
   IOField "I/O 域_2" at 383,410 size 35x48; FormatPattern 9
      ProcessValue <- "实际楼层数"
   IOField "I/O 域_3" at 415,278 size 35x48; FormatPattern 9
      ProcessValue <- "实际楼层数"
   IOField "I/O 域_4" at 415,152 size 35x48; FormatPattern 9
      ProcessValue <- "实际楼层数"
   IOField "I/O 域_5" at 379,20 size 35x48; FormatPattern 9
      ProcessValue <- "实际楼层数"
   Rectangle "矩形_3" at 659,6 size 127x38
      Appearance <- "开门步"
   TextField "文本域_7" at 673,125 size 77x27; Text '上行中'
   TextField "文本域_8" at 674,191 size 77x27; Text '下行中'
   TextField "文本域_9" at 599,331 size 70x68; Text '楼'
   Rectangle "矩形_6" at 750,124 size 39x35
      Appearance <- "上行"
   Rectangle "矩形_7" at 750,183 size 39x35
      Appearance <- "下行"
   Button "按钮_13" at 530,419 size 54x36; TextOff '启动'
      on Release: ResetBit("启动")
      on Press: SetBit("启动")
   Button "按钮_14" at 605,419 size 54x36; TextOff '停止'
      on Release: ResetBit("停止")
      on Press: SetBit("停止")
   Rectangle "矩形_8" at 609,456 size 50x20
      Appearance <- "停止指示灯"
   Rectangle "矩形_9" at 535,455 size 45x21
      Appearance <- "启动指示灯"
   Rectangle "矩形_10" at 91,355 size 65x108
      HorizontalMovement <- "门水平移动1"
   Rectangle "矩形_12" at 157,355 size 65x108
      HorizontalMovement <- "门水平移动1"
   Rectangle "矩形_11" at 91,240 size 65x108
      HorizontalMovement <- "门水平移动2"
   Rectangle "矩形_13" at 157,240 size 65x108
      HorizontalMovement <- "门水平移动2"
   Rectangle "矩形_14" at 93,125 size 65x108
      HorizontalMovement <- "门水平移动3"
   Rectangle "矩形_15" at 157,125 size 65x108
      HorizontalMovement <- "门水平移动3"
   Rectangle "矩形_16" at 92,10 size 65x108
      HorizontalMovement <- "门水平移动4"
   Rectangle "矩形_17" at 158,10 size 65x108
      HorizontalMovement <- "门水平移动4"
   Rectangle "矩形_1" at 100,400 size 115x58
      VerticalMovement <- "电梯位置"
*)